{attribute 'qualified_only'}
{attribute 'strict'}
TYPE E_LevelSensorID :
(
	Ch1_Rinse1 := 1,
    Ch2_Rinse2 := 2,
    Ch3_Rinse3 := 3,
    Ch4_Rinse4 := 4,
    Ch5_Waste  := 5
);
END_TYPE

(* stored: Version 1.1.0.1, ProductVersion 3.1.4024.12
   DUT E_LevelSensorID: Id {89bff82a-ccb0-43d9-9997-9e865835238a} *)
